// TIA Portal V20 export
TYPE "typeUnitCommunicationControlNodeBA030"
// stored: Namespace Unit1.Em0
   STRUCT
      noInterference { ExternalWritable := 'False'} : Bool;
      partClamped { ExternalWritable := 'False'} : Bool;
      partUnclamped { ExternalWritable := 'False'} : Bool;
      ngPartReady { ExternalWritable := 'False'} : Bool;
      ngLoadComplete { ExternalWritable := 'False'} : Bool;
   END_STRUCT;
END_TYPE
